{attribute 'linkalways'} 
{attribute 'no_explicit_call' := 'This FB is a CLASS and must be accessed using methods or properties'}
{attribute 'enable_dynamic_creation'}
FUNCTION_BLOCK FINAL GE_DINT EXTENDS Node
VAR
	in1 : _DINT(0);
	in2 : _DINT(0);
	out : _BOOL(FALSE);
END_VAR

METHOD PUBLIC Clone : I_Node
VAR
	pNode : POINTER TO GE_DINT;
END_VAR
pNode := __NEW(GE_DINT);
Clone := pNode^;
END_METHOD

METHOD FB_init : BOOL
VAR_INPUT
	bInitRetains : BOOL; // if TRUE, the retain variables are initialized (warm start / cold start)
	bInCopyCode : BOOL;  // if TRUE, the instance afterwards gets moved into the copy code (online change)
END_VAR
AddInput('in1',THIS^.in1);
AddInput('in2',THIS^.in2);
AddOutput('out', THIS^.out);
END_METHOD

METHOD PROTECTED OnExecute
VAR
END_VAR
out.Value := in1.Value >= in2.Value;
END_METHOD

END_FUNCTION_BLOCK

(* stored: Version 1.1.0.1, ProductVersion 3.1.4024.15
   POU GE_DINT: Id {03213b70-9564-42f4-8ac8-3d7c569c0f03}, SpecialFunc None
   Folder Constructor: Id {1388f8cb-5784-4bd1-b362-d010beb8c666}
   Method Clone: Id {ba4d4c44-c1da-4ef0-987c-f5fff2b6ab15}
   Method FB_init: Id {647c088c-3067-4722-8352-1750db09898c}
   Method OnExecute: Id {7dde363b-148c-4fca-b2f0-99c88ab4f8f5} *)
